{attribute addProperty BoxType "EK1100-0000-0018"}
{attribute addProperty Id "Beckhoff_EPP6xxxEK1122Beckhoff_EPP6xxxEK1122_B0D0374A5344668"}
{attribute addProperty CRC "2614931663"}
{attribute addProperty SizeInBites "5344"}
{attribute addProperty SizeInBytes "668"}
TYPE Beckhoff_EPP6xxx_9BDCB0CF EXTENDS EK1100_179A0949 :
STRUCT
	{attribute addProperty Name "Beckhoff_EPP6xxxEK1122"}
	Beckhoff_EPP6xxxEK1122 : Beckhoff_EPP6xxxEK1122_B0D0374A;
END_STRUCT
END_TYPE

(* stored: Version 1.2.0.0, ProductVersion 3.1.4024.9
   DUT Beckhoff_EPP6xxx_9BDCB0CF: Id {a0cabeb7-7547-47ed-957e-028192bfb165} *)
